FUNCTION_BLOCK StateComplete EXTENDS _AbstractState
VAR_INPUT
END_VAR
VAR_OUTPUT
END_VAR

(*
Determines whether the state can be activated.  
Returns `TRUE` by default but can be overridden for specific activation conditions.
*)
METHOD PROTECTED CanActivate : BOOL
CanActivate := _ctx.smgr.Current.Tag = _ctx.execute.Tag;
END_METHOD

(*
Executed when the state is entered.  
Provides a hook for defining state-specific behavior to be performed during the transition into this state.
*)
METHOD PROTECTED OnEntry
_ctx.sHmiStatusText := 'Complete: Next task please!';
END_METHOD

(*
Executed during the state's operation.  
Used to define state-specific logic that runs while the state is active.
*)
METHOD PROTECTED OnExecute
VAR
	strb: Strb;
END_VAR
IF _ctx.bHmiAcknowledge THEN	
	_ctx.smgr.Request(_ctx.idle);
END_IF
END_METHOD

END_FUNCTION_BLOCK

(* stored: Version 1.1.0.1
   POU StateComplete: Id {70ec6bcf-c012-4c5a-89e2-79b9d732c811}, SpecialFunc None
   Method CanActivate: Id {8c4689e7-3c91-4b2f-b68a-97b784123f6e}
   Method OnEntry: Id {f6cbc5dc-51f2-45cd-b81a-a21762d47304}
   Method OnExecute: Id {7b2f82b6-413f-44f8-a5cf-8013e51628f4} *)
